FUNCTION_BLOCK COMMUNICATION
VAR_INPUT
	
END_VAR
VAR_OUTPUT
END_VAR
VAR
	m_COMMUNICATION_MODE : COM_MODE;
	messageCreator : MESSAGE_CREATOR('CRISTART', 'CRIEND', 1);
	messageHandler : MESSAGE_HANDLER();
END_VAR

PROPERTY PUBLIC COMMUNICATION_MODE : COM_MODE
GET
COMMUNICATION_MODE := m_COMMUNICATION_MODE;
END_GET
SET
m_COMMUNICATION_MODE := COMMUNICATION_MODE;
END_SET
END_PROPERTY

METHOD PUBLIC CREATE : STRING
VAR_INPUT
	COMMAND : STRING;
	COMMAND_DETAILS : STRING;
END_VAR
VAR_OUTPUT
	ERROR : INT := 0;
END_VAR
IF (COMMUNICATION_MODE = COM_MODE.Robot) THEN 
	// creates string for robot when in Robot mode
	CREATE := MessageCreator.ROBOT_MESSAGE(COMMAND, COMMAND_DETAILS, ERROR => ERROR);
ELSIF (COMMUNICATION_MODE = COM_MODE.Monarco) THEN 
	// creates string for monarco when in Monarco mode
	CREATE := MessageCreator.MONARCO_MESSAGE_CMD(COMMAND_DETAILS, ERROR => ERROR);
			// JUST THE CMD MONARCO MESSAGE FOR NOW!!
END_IF
END_METHOD

METHOD FB_init : BOOL
VAR_INPUT
	bInitRetains : BOOL; // if TRUE, the retain variables are initialized (warm start / cold start)
	bInCopyCode : BOOL;  // if TRUE, the instance afterwards gets moved into the copy code (online change)
	
	communicationMODE : COM_MODE;
END_VAR
COMMUNICATION_MODE := communicationMode;
END_METHOD

METHOD PUBLIC HANDLE : INT
VAR_INPUT
	FULL_STRING : STRING;
END_VAR
IF (COMMUNICATION_MODE = COM_MODE.Robot) THEN 
	// handles string from robot when in Robot mode (RECEIVE_ROBOT())
	MessageHandler.RECEIVE_ROBOT(FULL_STRING, ERROR => HANDLE);
ELSIF (COMMUNICATION_MODE = COM_MODE.Monarco) THEN 
	// handles string from monarco when in Monarco mode (RECEIVE_MONARCO())
	MessageHandler.RECEIVE_MONARCO(FULL_STRING, ERROR => HANDLE);
END_IF
END_METHOD

END_FUNCTION_BLOCK

(* stored: Version 1.1.0.1, ProductVersion 3.1.4024.12
   POU COMMUNICATION: Id {ace835ab-6df9-403e-9e31-70d285ab16fc}, SpecialFunc None
   Property COMMUNICATION_MODE: Id {b296671c-fe1c-4ee7-8921-3f13e91d45b3}
   Get Get: Id {e6a11c6b-47d0-42f4-9fb5-2dd81a4fb2b8}
   Set Set: Id {49c2585b-4772-417f-bad3-17d38100fc36}
   Method CREATE: Id {aafc5eb4-35e9-4c88-b5bf-9f7dedabb599}
   Method FB_init: Id {5e0bba7a-d59d-4bdc-9140-ea6aebe74734}
   Method HANDLE: Id {e88f222e-5f0f-4f4e-a251-c44dcb49e058} *)
